FUNCTION_BLOCK FB_Panel
VAR_INPUT
	Modo: E_GEMMA;
	TR: TIME := T#3S; 	// Tiempo de reinicio
END_VAR

VAR_OUTPUT	
    Emergencia: BOOL; 	// := PE 				Parada de emergencia (seta)
 
						// POC - 				Conmutador PO Conectada  (negra)
	Marcha: BOOL; 		// :=FP_PM.Q 			Pulsador de marcha (verde)
    Reinicia: BOOL; 	// :=T(PM AND NOT PS) 	Restablece situacion inicial
	Restablece: BOOL;	// :=PM					Restablece la condición de fallo
	Restaura: BOOL;		// :=PM					Restaura condiciones iniciales
	
	Para: BOOL; 		// :=NOT PS				Pulsador de parada (rojo)
    Manual: BOOL; 		// :=SM			Conmutador de automático/manual (negro)
						// Pulsador de reset (azul)												

	// variables relacionadas con las pruebas de desarrollo
	Probando:	BOOL;	// DESDE LA VISU		Vamos a hacer pruebas
	ProbarExecute: 	BOOL;
	ProbarAck: BOOL;
	
	
	ProbarAlimentador: BOOL;
	ProbarCarga: BOOL;
	ProbarMedidor: BOOL;
	ProbarFotoelectrico: BOOL;
	ProbarInductivo: BOOL;
	ProbarEvacuador: BOOL;
	ProbarDescarga: BOOL;
	ProbarPlato: BOOL;
	ProbarNegarSensores: BOOL;
	FlancoNegarSensores: BOOL;
	
END_VAR
VAR
END_VAR

// pendiente vincular y codificar

END_FUNCTION_BLOCK

(* stored: Version 1.1.0.1, ProductVersion 3.1.4024.11
   POU FB_Panel: Id {514e5db3-ac71-4add-977b-df9fa295436c}, SpecialFunc None *)
